FUNCTION_BLOCK FB_HwRefInterlockSimple EXTENDS FB_HwRefInterlockBase
VAR
	bInput 	AT %I* : BOOL;
	bOutput AT %Q* : BOOL;
	nState : USINT;
	pXYDrive : POINTER TO FB_XYDriveBase;
END_VAR
VAR_OUTPUT
	
END_VAR

//Überwachung der Verriegelung
//Wenn Verriegelung durch Schlüssel oder mit Gewalt geöffnet wird, dann müssen die Antriebe
//gestoppt werden -> QuickStop -> PowerOFF
//QuickStop nur wenn Motion aktiv

CASE nState OF
	0:	//Überwachung im verriegelten Zustand
		IF NOT bInput THEN
			eCurrentState := E_InterlockState.Unlocked;
			fbXYDriveList.M_SetCurrentToHead();
			REPEAT
				pXYDrive := fbXYDriveList.M_Get();
				IF pXYDrive > 0 THEN
					pXYDrive^.M_Stop();
				END_IF
			UNTIL pXYDrive = 0
			END_REPEAT			
			nState := 1;
		END_IF
	1:
		fbXYDriveList.M_SetCurrentToHead();
		REPEAT
			pXYDrive := fbXYDriveList.M_Get();
			IF pXYDrive > 0 THEN
				pXYDrive^.M_PowerOff();
			END_IF
		UNTIL pXYDrive = 0
		END_REPEAT			
	
	10:	//Verriegeln
		//Unter welchen Bedingungen darf verrieglt werden?
		IF bInput THEN
			eCurrentState := E_InterlockState.Locked;
			nState := 0;
			fbXYDriveList.M_SetCurrentToHead();
			REPEAT
				pXYDrive := fbXYDriveList.M_Get();
				IF pXYDrive > 0 THEN
					IF pXYDrive^.P_bHomed AND NOT pXYDrive^.P_bError THEN
						pXYDrive^.M_PowerOn();
					END_IF
 				END_IF
			UNTIL pXYDrive = 0
			END_REPEAT			
		END_IF
	
	20: //Entriegelt
END_CASE

METHOD FB_init : BOOL
VAR_INPUT
	bInitRetains : BOOL; // if TRUE, the retain variables are initialized (warm start / cold start)
	bInCopyCode : BOOL;  // if TRUE, the instance afterwards gets moved into the copy code (online change)
END_VAR
eCurrentState := E_InterlockState.Locked;
END_METHOD

METHOD M_LockUnlock : ERRORID
VAR_INPUT
	bLock : BOOL;
END_VAR
IF bLock THEN	//Verriegln
	//IF eCurrentState 
	bOutput := FALSE;
	nState := 10;
ELSE	//Entriegeln
	//nur möglich, wenn keine manuelle Bewegung stattfindet
	IF MainDispacher.P_bReadyToUnlock THEN
		//bLocked := FALSE;
		bOutput := TRUE;	
	ELSE
		M_LockUnlock := E_ErrorIdCmd.ERRORID_NotReadyToUnlock;
	END_IF
END_IF
END_METHOD

END_FUNCTION_BLOCK

(* stored: Version 1.1.0.1, ProductVersion 3.1.4022.10
   POU FB_HwRefInterlockSimple: Id {79c1888d-719b-4736-adcd-b8d953d16a61}, SpecialFunc None
   Method FB_init: Id {a34f43ee-ffec-41c8-a8dc-ed95319ffac5}
   Method M_LockUnlock: Id {1f0c9354-7ec9-4a1a-8cc0-f9a8e18a2fb0} *)
